FUNCTION_BLOCK DST_RQST (* Concatenates management command DST and RQST fields *)
  (* Standard: 61499-1 *)
  (* Version 0.0, 2007-12-14, JHC, Holobloc Inc *)
  (* Compiler header: package fb.rt.ita; *)
  (* Compiler classdef: SimpleFB *)
  (* Compiler Java Sun JDK 1.5.0 *)
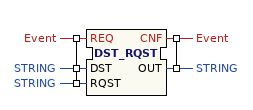
  EVENT_INPUT
    REQ WITH DST, RQST; (* Normal Execution Request *)
  END_EVENT
  EVENT_OUTPUT
    CNF WITH OUT; (* Execution Confirmation *)
  END_EVENT
  VAR_INPUT
    DST : STRING; (* Destination name *)
    RQST : STRING; (* Management request *)
  END_VAR
  VAR_OUTPUT
    OUT : STRING; (* DST '.' RQST *)
  END_VAR
  ALGORITHM REQ IN Java: (* Normally executed algorithm *)
OUT.length = DST.length + RQST.length + 1;
OUT.value = new byte[OUT.length];
System.arraycopy(DST.value,0,OUT.value,0,DST.length);
OUT.value[DST.length] = (byte)':';
System.arraycopy(RQST.value,0,OUT.value,DST.length+1,RQST.length);
  END_ALGORITHM
END_FUNCTION_BLOCK
